FUNCTION_BLOCK WaterTankSystem
  (* Standard: 61499-2 *)
  (* Version 0.1, 2015-00-11, syy, syy-PC *)
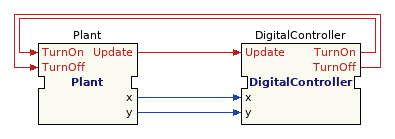
  FBS
    DigitalController : DigitalController;
    Plant : Plant;
  END_FBS
  EVENT_CONNECTIONS
    DigitalController.TurnOn TO Plant.TurnOn;
    DigitalController.TurnOff TO Plant.TurnOff;
    Plant.Update TO DigitalController.Update;
  END_CONNECTIONS
  DATA_CONNECTIONS
    Plant.x TO DigitalController.x;
    Plant.y TO DigitalController.y;
  END_CONNECTIONS
END_FUNCTION_BLOCK
